// SIMATIC S7-200 project (STEP 7-Micro/WIN), CPU 224 REL 02.01

SYMBOL_TABLE USER1
RUN              Q0.0
DIR              Q0.1
PB01             I0.0
PB02             I0.1
PB03             I0.2
S1               I0.3
S2               I0.4
S3               I0.5
END_SYMBOL_TABLE

ORGANIZATION_BLOCK MAIN:OB1
TITLE=PROGRAM COMMENTS
BEGIN
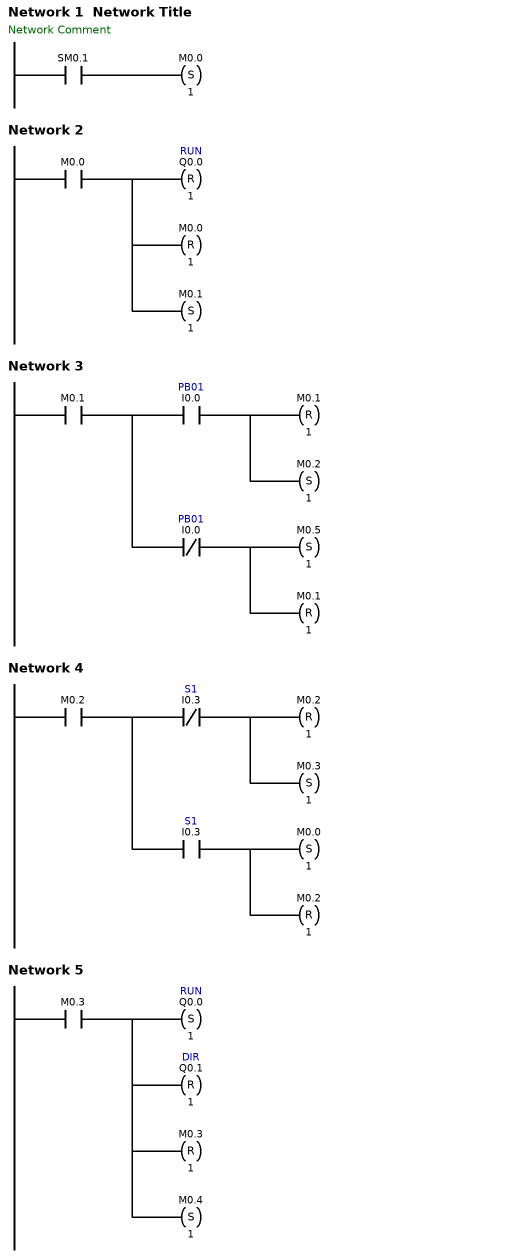
Network 1 // Network Title
// Network Comment
LD     SM0.1
S      M0.0, 1
Network 2
LD     M0.0
R      RUN:Q0.0, 1
R      M0.0, 1
S      M0.1, 1
Network 3
LD     M0.1
LPS
A      PB01:I0.0
R      M0.1, 1
S      M0.2, 1
LPP
AN     PB01:I0.0
S      M0.5, 1
R      M0.1, 1
Network 4
LD     M0.2
LPS
AN     S1:I0.3
R      M0.2, 1
S      M0.3, 1
LPP
A      S1:I0.3
S      M0.0, 1
R      M0.2, 1
Network 5
LD     M0.3
S      RUN:Q0.0, 1
R      DIR:Q0.1, 1
R      M0.3, 1
S      M0.4, 1
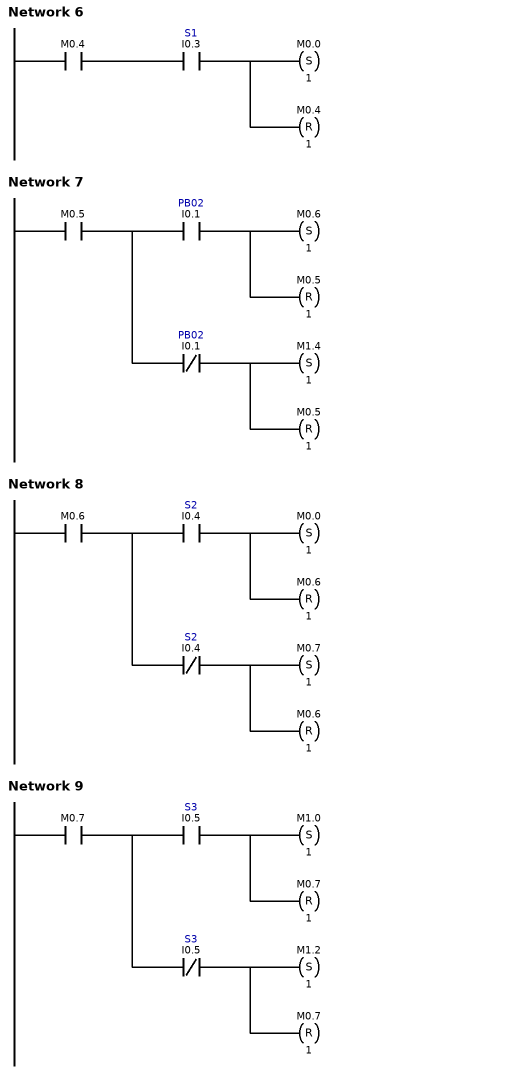
Network 6
LD     M0.4
A      S1:I0.3
S      M0.0, 1
R      M0.4, 1
Network 7
LD     M0.5
LPS
A      PB02:I0.1
S      M0.6, 1
R      M0.5, 1
LPP
AN     PB02:I0.1
S      M1.4, 1
R      M0.5, 1
Network 8
LD     M0.6
LPS
A      S2:I0.4
S      M0.0, 1
R      M0.6, 1
LPP
AN     S2:I0.4
S      M0.7, 1
R      M0.6, 1
Network 9
LD     M0.7
LPS
A      S3:I0.5
S      M1.0, 1
R      M0.7, 1
LPP
AN     S3:I0.5
S      M1.2, 1
R      M0.7, 1
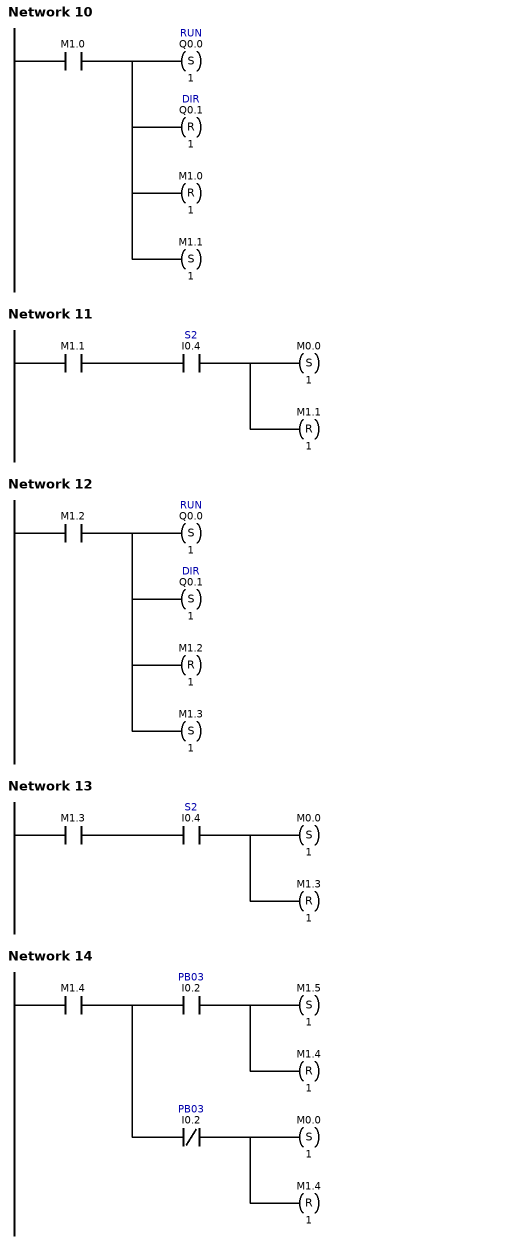
Network 10
LD     M1.0
S      RUN:Q0.0, 1
R      DIR:Q0.1, 1
R      M1.0, 1
S      M1.1, 1
Network 11
LD     M1.1
A      S2:I0.4
S      M0.0, 1
R      M1.1, 1
Network 12
LD     M1.2
S      RUN:Q0.0, 1
S      DIR:Q0.1, 1
R      M1.2, 1
S      M1.3, 1
Network 13
LD     M1.3
A      S2:I0.4
S      M0.0, 1
R      M1.3, 1
Network 14
LD     M1.4
LPS
A      PB03:I0.2
S      M1.5, 1
R      M1.4, 1
LPP
AN     PB03:I0.2
S      M0.0, 1
R      M1.4, 1
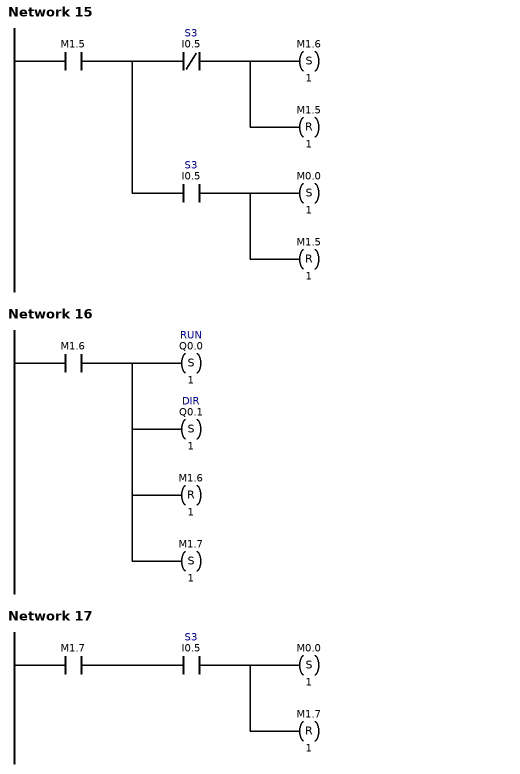
Network 15
LD     M1.5
LPS
AN     S3:I0.5
S      M1.6, 1
R      M1.5, 1
LPP
A      S3:I0.5
S      M0.0, 1
R      M1.5, 1
Network 16
LD     M1.6
S      RUN:Q0.0, 1
S      DIR:Q0.1, 1
R      M1.6, 1
S      M1.7, 1
Network 17
LD     M1.7
A      S3:I0.5
S      M0.0, 1
R      M1.7, 1
END_ORGANIZATION_BLOCK
